// Mitsubishi GX Works2 project: halvanika_new3   PLC: FX3U/FX3UC

TYPE vat : STRUCT
  entire : INT;
  prioriyry : BOOL;
  timer_s : DINT;
  on_off : BOOL;
  timer_off : BOOL;
  timer_real : DINT;
  vibor : INT;
  air_off : BOOL;
  vanna_off : BOOL;
END_STRUCT END_TYPE

// global labels: Global1
VAR_GLOBAL
  incFR AT D100 : INT;  (* позиция балки по ваннам *)
  incUD AT D101 : INT;  (* позиция балки по вертикали *)
  muving AT D102 : INT;  (* управление с HMI балкой *)
  Program_exec AT D103 : INT;  (* переключение режимов работы *)
  tub : ARRAY [0..15] OF vat;  (* массив структуры ванн *)
  init_reset AT M100 : BOOL;  (* переключение инициализации *)
  autoStop AT D104 : INT;  (* включение окна ошибок *)
  text AT D105 : STRING[32];  (* Сообщения об ошибках *)
  TEST_ONOFF AT D107 : INT;  (* Тестовое отключение бурбуляторов *)
  Hide_button AT D108 : INT;
  temper AT D110 : ARRAY [0..8] OF INT;
  load_z AT D120 : INT;
  upload_z AT D121 : INT;
  init_move : BOOL;
  reset_timers : BOOL;
  pause AT D122 : INT;
  blink_botton AT D123 : INT;
  ch AT D124 : INT;
END_VAR

// task Task_01 (event TRUE, interval 0, priority 31): Init

PROGRAM Init
VAR
  Manual_1 : Manual;
  Auto_1 : Auto;
  Reset_1 : Reset;
  init : BOOL;
  Stop_program : BOOL;
  Count : INT;
  blink : TON;
  TR1 : R_TRIG;
  Count2 : INT;
  bath_02 : TON;
  bath_03 : TON;
  bath_04 : TON;
  bath_05 : TON;
  bath_06 : TON;
  bath_07 : TON;
  bath_08 : TON;
  bath_09 : TON;
  bath_10 : TON;
  bath_11 : TON;
  bath_12 : TON;
  bath_13 : TON;
  bath_14 : TON;
END_VAR
(*------------------------------INIT----------------------------------------------------*)
IF NOT init THEN
	incFR := 1;
	incUD := -1;
	Hide_button := 1;
	Program_exec := 0;
	muving := 0;
	TEST_ONOFF :=1;
reset_timers := FALSE;
pause := 0;
blink_botton := 0;

	tub[1].prioriyry := 0;
	tub[2].prioriyry := 1;
	tub[3].prioriyry := 0;
	tub[4].prioriyry := 0;
	tub[5].prioriyry := 1;
	tub[6].prioriyry := 0;
	tub[7].prioriyry := 0;
	tub[8].prioriyry := 1;
	tub[9].prioriyry := 0;
	tub[10].prioriyry := 1;
	tub[11].prioriyry := 1;
	tub[12].prioriyry := 0;
	tub[13].prioriyry := 0;
	tub[14].prioriyry := 1;
	tub[15].prioriyry := 1;
	
		FOR Count := 1 TO 15 DO
			tub[Count].vanna_off := 1;
			tub[Count].air_off := 0;
		END_FOR;	
	
	init := TRUE;
END_IF;

(*------------------------------PROGAM----------------------------------------------------*)

IF (X000 = 0) AND (X001 = 1) AND (X002 = 1) THEN incFR := 1;  END_IF;
IF (X000 = 1) AND (X001 = 1) AND (X002 = 1) THEN incFR := 15; END_IF;
IF (X004 = 1)  THEN incUD := -1; ELSIF  (X003 = 1) THEN  incUD := 1;  END_IF;
IF incFR < 1 OR incFR > 15 THEN autoStop := 1; END_IF;
	
(*------------------------------Timers----------------------------------------------------*)

	FOR count:=2 TO 14 DO
		IF NOT tub[Count].timer_off THEN tub[Count].timer_real:=0; END_IF;
	END_FOR;
	
IF Program_exec <> 3 THEN	
bath_02(IN:= INT_TO_BOOL(tub[2].entire) ,PT:= DINT_TO_TIME(tub[2].timer_s) * 1000);
bath_03(IN:= INT_TO_BOOL(tub[3].entire) ,PT:= DINT_TO_TIME(tub[3].timer_s) * 1000);
bath_04(IN:= INT_TO_BOOL(tub[4].entire) ,PT:= DINT_TO_TIME(tub[4].timer_s) * 1000);
bath_05(IN:= INT_TO_BOOL(tub[5].entire) ,PT:= DINT_TO_TIME(tub[5].timer_s) * 1000);
bath_06(IN:= INT_TO_BOOL(tub[6].entire) ,PT:= DINT_TO_TIME(tub[6].timer_s) * 1000);
bath_07(IN:= INT_TO_BOOL(tub[7].entire) ,PT:= DINT_TO_TIME(tub[7].timer_s) * 1000);
bath_08(IN:= INT_TO_BOOL(tub[8].entire) ,PT:= DINT_TO_TIME(tub[8].timer_s) * 1000);
bath_09(IN:= INT_TO_BOOL(tub[9].entire) ,PT:= DINT_TO_TIME(tub[9].timer_s) * 1000);
bath_10(IN:= INT_TO_BOOL(tub[10].entire) ,PT:= DINT_TO_TIME(tub[10].timer_s) * 1000);
bath_11(IN:= INT_TO_BOOL(tub[11].entire) ,PT:= DINT_TO_TIME(tub[11].timer_s) * 1000);
bath_12(IN:= INT_TO_BOOL(tub[12].entire) ,PT:= DINT_TO_TIME(tub[12].timer_s) * 1000);
bath_13(IN:= INT_TO_BOOL(tub[13].entire) ,PT:= DINT_TO_TIME(tub[13].timer_s) * 1000);
bath_14(IN:= INT_TO_BOOL(tub[14].entire) ,PT:= DINT_TO_TIME(tub[14].timer_s) * 1000);

tub[2].timer_off := NOT bath_02.Q; tub[2].timer_real := TIME_TO_DINT(bath_02.ET) / 1000;
tub[3].timer_off := NOT bath_03.Q; tub[3].timer_real := TIME_TO_DINT(bath_03.ET) / 1000;
tub[4].timer_off := NOT bath_04.Q; tub[4].timer_real := TIME_TO_DINT(bath_04.ET) / 1000;
tub[5].timer_off := NOT bath_05.Q; tub[5].timer_real := TIME_TO_DINT(bath_05.ET) / 1000;
tub[6].timer_off := NOT bath_06.Q; tub[6].timer_real := TIME_TO_DINT(bath_06.ET) / 1000;
tub[7].timer_off := NOT bath_07.Q; tub[7].timer_real := TIME_TO_DINT(bath_07.ET) / 1000;
tub[8].timer_off := NOT bath_08.Q; tub[8].timer_real := TIME_TO_DINT(bath_08.ET) / 1000;
tub[9].timer_off := NOT bath_09.Q; tub[9].timer_real := TIME_TO_DINT(bath_09.ET) / 1000;
tub[10].timer_off := NOT bath_10.Q; tub[10].timer_real := TIME_TO_DINT(bath_10.ET) / 1000;
tub[11].timer_off := NOT bath_11.Q; tub[11].timer_real := TIME_TO_DINT(bath_11.ET) / 1000;
tub[12].timer_off := NOT bath_12.Q; tub[12].timer_real := TIME_TO_DINT(bath_12.ET) / 1000;
tub[13].timer_off := NOT bath_13.Q; tub[13].timer_real := TIME_TO_DINT(bath_13.ET) / 1000;
tub[14].timer_off := NOT bath_14.Q; tub[14].timer_real := TIME_TO_DINT(bath_14.ET) / 1000;

(* Включить ток*);
IF tub[5].entire = 1 THEN Y013 := INT_TO_BOOL(TEST_ONOFF); END_IF;
IF tub[10].entire = 1 THEN Y024 :=  INT_TO_BOOL(TEST_ONOFF); END_IF;
IF tub[11].entire = 1 THEN Y014 :=  INT_TO_BOOL(TEST_ONOFF); END_IF;
(* Выключить ток*);
IF NOT tub[5].timer_off THEN Y013 := 0; END_IF;
IF NOT tub[10].timer_off THEN Y024 := 0; END_IF;
IF NOT tub[11].timer_off THEN Y014 := 0; END_IF;
	
(* Включить спрей*)
IF tub[3].on_off THEN Y016 := INT_TO_BOOL(TEST_ONOFF); ELSE Y016 := FALSE; END_IF;
IF tub[6].on_off THEN Y017 :=  INT_TO_BOOL(TEST_ONOFF); ELSE Y017 := FALSE; END_IF;
IF tub[9].on_off THEN Y020 :=  INT_TO_BOOL(TEST_ONOFF); ELSE Y020 := FALSE; END_IF;
IF tub[12].on_off THEN Y021 :=  INT_TO_BOOL(TEST_ONOFF); ELSE Y021 := FALSE; END_IF;

(* Включить спрей
IF tub[3].entire = 1 THEN Y016 :=  INT_TO_BOOL(TEST_ONOFF); END_IF;
IF tub[6].entire = 1 THEN Y017 :=  INT_TO_BOOL(TEST_ONOFF); END_IF;
IF tub[9].entire = 1 THEN Y020 :=  INT_TO_BOOL(TEST_ONOFF); END_IF;
IF tub[12].entire = 1 THEN Y021 :=  INT_TO_BOOL(TEST_ONOFF); END_IF;

Выключить спрей
IF NOT tub[3].timer_off THEN Y016 := 0; END_IF;
IF NOT tub[6].timer_off THEN Y017 := 0; END_IF;
IF NOT tub[9].timer_off THEN Y020 := 0; END_IF;
IF NOT tub[12].timer_off THEN Y021 := 0; END_IF;
	
Выключить сушку
IF NOT tub[14].timer_off THEN Y011 := 0;  END_IF; 
*);
END_IF;

IF reset_timers THEN
	bath_02(IN:= FALSE);
	bath_03(IN:= FALSE);
	bath_04(IN:= FALSE);
	bath_05(IN:= FALSE);
	bath_06(IN:= FALSE);
	bath_07(IN:= FALSE);
	bath_08(IN:= FALSE);
	bath_09(IN:= FALSE);
	bath_10(IN:= FALSE);
	bath_11(IN:= FALSE);
	bath_12(IN:= FALSE);
	bath_13(IN:= FALSE);
	bath_14(IN:= FALSE);
	reset_timers := FALSE;
END_IF;

(*------------------------------CASE----------------------------------------------------*)

IF pause = 0 AND (Program_exec = 1 OR  (X011 = 1)) THEN
	Manual_1(); 
	
ELSIF Program_exec = 2 THEN
	Auto_1(); 
	(* -------------Air Pump----------*)
	Y030 := tub[2].air_off;
	Y031 := tub[3].air_off;
	Y032 := tub[4].air_off;
	Y033 := tub[5].air_off;
	Y034 := tub[6].air_off;
	Y035 := tub[7].air_off;
	Y036 := tub[8].air_off;
	Y037 := tub[9].air_off;
	Y040 := tub[10].air_off;
	Y041 := tub[11].air_off;
	Y042 := tub[12].air_off;
	Y043 := tub[13].air_off;
	
ELSIF Program_exec = 3 THEN
	Reset_1();
	reset_timers := TRUE;
END_IF;

IF pause = 1 AND (Program_exec = 1 OR  (X011 = 1)) THEN
	Program_exec := 2;
	pause := 2;
	END_IF;
muving := 0;


(*------------------------------STOP----------------------------------------------------*)

IF (X013 = 1) OR (X021 = 1) OR (X012 = 1)  OR autoStop = 1THEN
	Program_exec := 0;
	muving := 0;
	autoStop := 0;
	Hide_button := 0;
	pause := 0;

	Y000 :=0;	Y010 :=0;	Y020 :=0;
	Y001 :=0;	Y011 :=0;	Y021 :=0;
	Y002 :=0;	Y012 :=0;	Y022 :=0;
	Y003 :=0;	Y013 :=0;	Y023 :=0;
	Y004 :=0;	Y014 :=0;	Y024 :=0;
	Y005 :=0;	Y015 :=0;	Y025 :=0;
	Y006 :=0;	Y016 :=0;	Y026 :=0;
	Y007 :=0;	Y017 :=0;	Y027 :=0;
		(* -------------Air Pump----------*)
	Y030 := 0;	Y040 := 0;
	Y031 := 0;	Y041 := 0;
	Y032 := 0;	Y042 := 0;
	Y033 := 0;	Y043 := 0;
	Y034 := 0;	Y044 := 0;
	Y035 := 0;	Y045 := 0;
	Y036 := 0;	Y046 := 0;
	Y037 := 0;	Y047 := 0;
	
	reset_timers := TRUE;
	
		FOR Count := 1 TO 15 DO
			tub[Count].timer_off  := 0;
			tub[Count].timer_real := 0;
			tub[Count].on_off := 0;
			tub[Count].air_off := 0;
		END_FOR;	
		
		init_move:= FALSE; 
		init_reset := FALSE;
		

END_IF;
END_PROGRAM

FUNCTION_BLOCK Auto
VAR
  blink : TON;
  init : BOOL;
  vanna : INT;
  Count : INT;
  vanna1 : INT;
  tabs : INT;
  TR1 : R_TRIG;
  Err : INT;
  prime : BOOL;
  vanna15 : INT;
  moving_1 : moving;
  pause_t : TON;
  TR2 : R_TRIG;
  stopd : BOOL;
  vanOff : INT;
  Counts : INT;
END_VAR
(*------------------------------INIT----------------------------------------------------*)
IF NOT init_reset THEN
	text:= "";
	IF incUD = 1 THEN text:= "Lower the beam down"; Program_exec := 0; END_IF; 
		vanna1 := 0;
		vanna := 0;
		vanna15 := 0;
		pause := 1;
		stopd := FALSE;
		ch := 1;
		vanOff := 1;
		(*Doors close*)
		Y022 := 0;
		blink_botton := 2;
		pause_t(IN := FALSE);
		TR2(_CLK := FALSE);
	init_reset :=TRUE;
	
END_IF;


(*------------------------------Blink----------------------------------------------------*)
Y026:= 0;
blink(IN:= NOT blink.Q, PT:= T#1s);
TR1(_CLK:= blink.Q );
IF TR1.Q THEN
	Y015:= NOT Y015;
	IF  tub[15].entire = 1 AND upload_z = 0 THEN Y027:= NOT Y027; ELSE Y027:= FALSE; END_IF;
END_IF;

(*------------------------------Blink----------------------------------------------------*)

pause_t (IN:= stopd, PT:= T#4s);
TR2(_CLK:= pause_t.Q );
IF TR2.Q THEN
	tabs:= tabs +1;
	stopd := FALSE;
END_IF;

(*-----------------------------CICLE-----------------------------------------------------*)


IF X006 = 1 OR upload_z = 1 THEN vanna15 := 15; upload_z := 1; END_IF;
IF  X005 = 1 OR load_z = 1 THEN vanna1 := 1; tub[1].entire := 1; load_z := 1; END_IF;
	
IF vanna = 0 THEN
	prime := FALSE;
	tabs := 0;
	vanOff := 1;
	Counts := 0;
	
	FOR Count := 2 TO 14 BY 1 DO
		IF tub[Count].entire = 1 AND tub[Count+vanOff ].entire = 0 AND NOT tub[Count].timer_off AND NOT tub[Count].prioriyry AND NOT prime THEN vanna := Count; prime := FALSE;  END_IF;
		IF tub[Count].entire = 1 AND tub[Count+vanOff ].entire = 0 AND NOT tub[Count].timer_off AND tub[Count].prioriyry THEN vanna := Count; prime := TRUE; END_IF;
	END_FOR;	
	
	IF tub[1].entire =0 AND  vanna15 = 15 THEN vanna := vanna15; END_IF;
	IF tub[2].entire =0 AND vanna1 = 1 THEN vanna := vanna1; END_IF;
	
	FOR Count := vanna TO 14 DO
		IF tub[vanna+vanOff ].vanna_off = 0 THEN vanOff := vanOff + 1;
		ELSE
			EXIT;
		END_IF;
	END_FOR;
	 IF tub[vanna+vanOff].entire = 1 THEN vanna := 0; END_IF;
	
END_IF;
		
(*-----------------------------ERROR-----------------------------------------------------*)	
(*	Ошибки обрабатываем в HMI *)
(*-----------------------------ERROR-----------------------------------------------------*)		
	
	IF vanna > 0 AND tabs = 0 THEN			
				IF incFR > vanna THEN
					moving_1(mv:=  2 ,mv_change:= incFR - vanna ,incount:= incFR, incUP:= incUD, ends:= tabs);
				ELSIF  incFR < vanna THEN
					moving_1(mv:=  1 ,mv_change:= vanna - incFR ,incount:= incFR, incUP:= incUD, ends:= tabs);
				ELSE
					tabs:= 1;
				END_IF;
		
	ELSE
 
	    CASE vanna OF
	
			1:  IF tub[vanna+vanOff].entire = 0 THEN
			CASE tabs OF	
						1: moving_1(mv:=  3 ,mv_change:= 1 ,incount:= incFR, incUP:= incUD, ends:= tabs);
						2: IF TRUE THEN tub[vanna].entire := 0; tabs:= tabs+1; END_IF;
						3: tabs:= tabs +1;
						4: moving_1(mv:= 1 ,mv_change:= vanOff ,incount:= incFR, incUP:= incUD, ends:= tabs);
						5: IF TRUE THEN stopd := TRUE; tub[vanna+vanOff].air_off := TRUE; END_IF;
						6: moving_1(mv:=  4 ,mv_change:= 1 ,incount:= incFR, incUP:= incUD, ends:= tabs);
						7: tabs:= tabs +1;
						8: IF TRUE THEN
							tub[vanna+vanOff].entire := 1;
							tub[vanna+vanOff].timer_off := TRUE;
							vanna := 0;
							vanna1 := 0;
							tabs:= 0;
							END_IF;
			END_CASE;
			END_IF;
		
			3, 6, 9, 12:  IF TRUE THEN
			CASE tabs OF
						1: IF TRUE THEN tub[vanna].on_off := TRUE; tabs:= tabs+1; END_IF;	
						2: moving_1(mv:=  3 ,mv_change:= 1 ,incount:= incFR, incUP:= incUD, ends:= tabs);
						3: IF TRUE THEN tub[vanna].entire := 0; tub[vanna].air_off := FALSE; tub[vanna].on_off := FALSE; tabs:= tabs+1; END_IF;
						4: moving_1(mv:= 1 ,mv_change:= vanOff ,incount:= incFR, incUP:= incUD, ends:= tabs); 
						5: IF TRUE THEN stopd := TRUE; tub[vanna+vanOff].air_off := TRUE; END_IF;
						6: moving_1(mv:=  4 ,mv_change:= 1 ,incount:= incFR, incUP:= incUD, ends:= tabs);
						7: tabs:= tabs +1;
						8: IF TRUE THEN
								tub[vanna+vanOff].entire := 1;
								tub[vanna+vanOff].timer_off := TRUE;
								vanna := 0;
								tabs:= 0;
							END_IF;
			END_CASE;
			END_IF;
	
			2, 4, 5, 8, 10, 11:  IF TRUE THEN
			CASE tabs OF	
						1: moving_1(mv:=  3 ,mv_change:= 1 ,incount:= incFR, incUP:= incUD, ends:= tabs);
						2: IF TRUE THEN tub[vanna].entire := 0; tub[vanna].air_off := FALSE; tabs:= tabs+1; END_IF;
						3: tabs:= tabs +1;
						4: moving_1(mv:= 1 ,mv_change:= vanOff ,incount:= incFR, incUP:= incUD, ends:= tabs); 
						5: IF TRUE THEN stopd := TRUE; tub[vanna+vanOff].air_off := TRUE; END_IF;
						6: moving_1(mv:=  4 ,mv_change:= 1 ,incount:= incFR, incUP:= incUD, ends:= tabs);
						7: tabs:= tabs +1;
						8: IF TRUE THEN
							tub[vanna+vanOff].entire := 1;
							tub[vanna+vanOff].timer_off := TRUE;
								vanna := 0;
								tabs:= 0;
							END_IF;
			END_CASE;
			END_IF;
	
			7:  IF tub[vanna+vanOff +1].entire = 0 THEN
			CASE tabs OF	
						1: moving_1(mv:=  3 ,mv_change:= 1 ,incount:= incFR, incUP:= incUD, ends:= tabs);
						2: IF TRUE THEN tub[vanna].entire := 0; tub[vanna].air_off := FALSE; tabs:= tabs+1; END_IF;
						3: tabs:= tabs +1;
						4: moving_1(mv:= 1 ,mv_change:= vanOff ,incount:= incFR, incUP:= incUD, ends:= tabs); 
						5: IF TRUE THEN stopd := TRUE; tub[vanna+vanOff].air_off := TRUE; END_IF;
						6: moving_1(mv:=  4 ,mv_change:= 1 ,incount:= incFR, incUP:= incUD, ends:= tabs);
						7: tabs:= tabs +1;
						8: IF TRUE THEN
							tub[vanna+vanOff].entire := 1;
							tub[vanna+vanOff].timer_off := TRUE;
							tabs:=tabs+1;
							END_IF;
						9:	IF NOT tub[vanna+vanOff].timer_off  THEN
								vanna := vanna + 1;
								tabs:= 0;
							END_IF;
							
			END_CASE;
			END_IF;
	
			13:  IF TRUE THEN
			CASE tabs OF	
						1: moving_1(mv:=  3 ,mv_change:= 1 ,incount:= incFR, incUP:= incUD, ends:= tabs);
						2: IF TRUE THEN tub[vanna].entire := 0; tub[vanna].air_off := FALSE; tabs:= tabs+1; END_IF;
						3: tabs:= tabs +1;
						4: moving_1(mv:= 1 ,mv_change:= vanOff ,incount:= incFR, incUP:= incUD, ends:= tabs); 
						(*Doors open*)
						5: IF TRUE THEN Y022 := 1; tabs:= tabs+1; END_IF;
						6: moving_1(mv:=  4 ,mv_change:= 1 ,incount:= incFR, incUP:= incUD, ends:= tabs);
						7: tabs:= tabs +1;
						8: IF TRUE THEN
						(*Doors close*)
							Y022 := 0;
							tub[vanna+vanOff].entire := 1;
							tub[vanna+vanOff].timer_off := TRUE;
							vanna := 0;
							tabs:= 0;
							END_IF;
			END_CASE;
			END_IF;
			
			14:  IF TRUE THEN
			CASE tabs OF
						(*-Doors open-вернуться*)	
						1: IF TRUE THEN Y022 := 1; tabs:= tabs+1; END_IF;
						2: moving_1(mv:=  3 ,mv_change:= 1 ,incount:= incFR, incUP:= incUD, ends:= tabs);
						3: tabs:= tabs +1;
						4: IF TRUE THEN Y022:=0; tub[vanna].entire := 0; tabs:= tabs+1; END_IF;
						5: moving_1(mv:= 1 ,mv_change:= 1 ,incount:= incFR, incUP:= incUD, ends:= tabs);
						6: moving_1(mv:=  4 ,mv_change:= 1 ,incount:= incFR, incUP:= incUD, ends:= tabs);
						7: tabs:= tabs +1;
						8: IF TRUE THEN
							tub[vanna+1].entire := 1;
							tub[vanna+1].timer_off := TRUE;
							vanna := 0;
							tabs:= 0;
							END_IF;
			END_CASE;
			END_IF;
			
			15:  IF tub[1].entire = 0 THEN
			CASE tabs OF	
						1: moving_1(mv:=  3 ,mv_change:= 1 ,incount:= incFR, incUP:= incUD, ends:= tabs);
						2: IF TRUE THEN tub[vanna].entire := 0; tabs:= tabs+1; END_IF;
						3: moving_1(mv:= 2 ,mv_change:= 14 ,incount:= incFR, incUP:= incUD, ends:= tabs);
						4: moving_1(mv:=  4 ,mv_change:= 1 ,incount:= incFR, incUP:= incUD, ends:= tabs);
						5: tabs:= tabs +2;
						7: IF TRUE THEN
							vanna := 0;
							vanna15 :=0;
							tabs:= 0;
							END_IF;
			END_CASE;
			END_IF;
		
	    END_CASE;
    END_IF;

IF vanna = 0 AND pause = 2 THEN  pause := 0; Program_exec := 1; ELSE  Program_exec := 2;  END_IF;
END_FUNCTION_BLOCK

FUNCTION_BLOCK Manual
VAR
  blink : TON;
  TR1 : R_TRIG;
  tabs : INT;
  MV : INT;
  DELTA_MV : INT;
  moving_1 : moving;
END_VAR

Y015 := 0;
blink(IN:= NOT blink.Q, PT:= T#1s);
TR1(_CLK:= blink.Q );
IF TR1.Q THEN
	Y026:= NOT Y026;
END_IF;
pause := 0;
blink_botton := 1;
Program_exec := 1;
IF  (X001 = 0)  THEN ch:=0; ELSE ch:=1; END_IF;
DELTA_MV:= 1;
init_reset := FALSE;

	IF		((X005 = 1) OR (muving=1))  AND  (incFR < 15) THEN
		MV:= 1;					(* Forward *)
	ELSIF ((X006 = 1) OR (muving=2)) AND  (incFR > 1) THEN
		MV:= 2;						(* Revers *)
	ELSIF ((X007 = 1) OR (muving=3)) THEN
		MV:= 3;					(* Up *)
	ELSIF ((X010 = 1)  OR (muving=4)) THEN
		MV:= 4;						(* Down *)
	END_IF;
	moving_1(mv:=  MV, mv_change:= DELTA_MV, incount:= incFR, incUP:= incUD);
muving := 0;
MV:=0;
END_FUNCTION_BLOCK

FUNCTION_BLOCK Reset
VAR
  Count : INT;
  init : BOOL;
END_VAR
IF (X000 = 0) AND (X001 = 1) AND (X002 = 1) THEN incFR := 1; END_IF;
IF (X000 = 1) AND (X001 = 1) AND (X002 = 0) THEN incFR := 15; END_IF;
IF (X004 = 1)  THEN incUD := -1; ELSIF  (X003 = 1) THEN  incUD := 1;  END_IF;
	
(*------------------------------INIT----------------------------------------------------*)
	IF NOT init THEN 
	Y027 :=1;	
	Y000 :=0;	Y010 :=0;	Y020 :=0;
	Y001 :=0;	Y011 :=0;	Y021 :=0;
	Y002 :=0;	Y012 :=0;	Y022 :=0;
	Y003 :=0;	Y013 :=0;	Y023 :=0;
	Y004 :=0;	Y014 :=0;	Y024 :=0;
	Y005 :=0;	Y015 :=0;	Y025 :=0;
	Y006 :=0;	Y016 :=0;	Y026 :=0;
	Y007 :=0;	Y017 :=0;	
		(* -------------Air Pump----------*)
	Y030 := 0;	Y040 := 0;
	Y031 := 0;	Y041 := 0;
	Y032 := 0;	Y042 := 0;
	Y033 := 0;	Y043 := 0;
	Y034 := 0;	Y044 := 0;
	Y035 := 0;	Y045 := 0;
	Y036 := 0;	Y046 := 0;
	Y037 := 0;	Y047 := 0;
	
	tub[1].prioriyry := 0;
	tub[2].prioriyry := 1;
	tub[3].prioriyry := 0;
	tub[4].prioriyry := 0;
	tub[5].prioriyry := 1;
	tub[6].prioriyry := 0;
	tub[7].prioriyry := 0;
	tub[8].prioriyry := 1;
	tub[9].prioriyry := 0;
	tub[10].prioriyry := 1;
	tub[11].prioriyry := 1;
	tub[12].prioriyry := 0;
	tub[13].prioriyry := 0;
	tub[14].prioriyry := 1;
	tub[15].prioriyry := 1;
	
	muving := 0;
blink_botton := 3;
	init := TRUE; 
	END_IF;
	
	init_reset := FALSE;
	pause := 0;
	
	FOR Count := 1 TO 15 DO
		tub[Count].entire := 0;
		tub[Count].timer_off  := 0;
		tub[Count].timer_real:=0;
		tub[Count].on_off:=0;
		tub[Count].vanna_off := 1;
		tub[Count].air_off := 0;
	END_FOR;	
 
 (*IF X004 = 0 THEN moving_1(mv:=  4, mv_change:= 1, incount:= incFR, incUP:= incUD); END_IF;*)
 	
 	IF (X000 = 0) AND (X001 = 1) AND (X002 = 1) THEN
		Y000 := 0;
		Y001 := 0;
		Y002 := 0;
		Y003 := 0;
		Y004 := 0;
		incFR := 1; 
	Program_exec := 0;
		Y027 :=0;
 	ELSE
 		Y004 := 1;
		Y002 := 0;
		Y001 := 1;
		IF (X002 = 1) THEN Y003 := 0; 
		ELSIF (X001 = 1) AND (X002 = 0) THEN Y003 := 1; 
		END_IF;
		
END_IF;
END_FUNCTION_BLOCK

FUNCTION_BLOCK moving
VAR_INPUT
  mv : INT;
END_VAR
VAR
  flag : INT;
  temp : INT;
END_VAR
VAR_INPUT
  mv_change : INT;
END_VAR
VAR
  change : INT;
  beg : INT;
END_VAR
VAR_IN_OUT
  incount : INT;
END_VAR
VAR
  count : INT;
END_VAR
VAR_IN_OUT
  incUP : INT;
END_VAR
VAR_OUTPUT
  ends : INT;
END_VAR
VAR
  init : BOOL;
END_VAR
	(*------------------------------INIT----------------------------------------------------*)
IF NOT init_move THEN
	flag :=0;
	temp:=0;
	
				incount := incount;
			incUP:=incUP;
			beg:=1;

	init_move:=TRUE;
	END_IF;
	
	IF temp = 0  AND mv <> 0 AND mv_change <> 0 THEN
		flag := 1; 
		temp := mv;
		change := mv_change-ch; 
		ch:=1;
		beg := 1;

	END_IF;

	CASE temp OF
			1:		IF flag = 1 THEN 
						Y000 := 1;
						Y003 := 0;
						Y004 := 1;
					IF (X000 = 1) AND flag =1THEN change := change - beg; 
							incount := incount +beg;
							beg := 0;
							Y002 := 1;
						ELSE 
							beg :=1;
							 END_IF;
						IF change <= 0 THEN 	flag := 2; END_IF;
					ELSIF (X000 = 0) AND (X001 = 0) AND (X002 = 1) AND flag = 2  THEN
						Y003 := 1;
						Y002 := 0;	
				(*			REPEAT
								IF (X001 = 1) THEN change := change - 1; moveFR := 1;END_IF;
							UNTIL change = 0 END_REPEAT; *)
						flag := 3;
					ELSIF (X000 = 1) AND (X001 = 0) AND (X002 = 0)  AND flag = 3 THEN
						Y002 := 0;
						Y003 := 0;
						flag := 4;
					ELSIF (X001 = 1) AND (X002 = 0)  AND flag = 4  THEN
						Y000 := 0;
						Y002 := 0;
						Y003 := 0;
						flag := 0;
						temp := 0;
						Y004 := 0;
incount := incount+1;
ends:= 1+ends;
						END_IF;

			(*-----------------*)
			2:		IF flag = 1 THEN 
						Y001 := 1;
						Y003 := 0;
						Y004 := 1;
					IF (X002 = 1) AND flag =1THEN change := change - beg; 
							incount := incount -beg;
							beg := 0;
							Y002 := 1;
						ELSE 
							beg :=1;
							 END_IF;
						IF change <= 0 THEN 	flag := 2; END_IF;
					ELSIF  (X000 = 1) AND (X001 = 0) AND (X002 = 0)  AND flag = 2 THEN
						Y003 := 1;
						Y002 := 0;
						flag := 3;
					ELSIF (X000 = 0) AND (X001 = 0) AND (X002 = 1)   AND flag = 3 THEN
						Y002 := 0;
						Y003 := 0;
						flag := 4;
					ELSIF  (X000 = 0) AND (X001 = 1)  AND flag = 4  THEN
						Y001 := 0;
						Y002 := 0;
						Y003 := 0;
						flag := 0;
						temp := 0;
						Y004 := 0;
ends:= 1+ends;				
incount := incount-1;	
						END_IF;
						
						3:		IF  (X003 = 1) THEN 
						Y000 := 0;
						Y001 := 0;
						Y002 := 0;
						Y003 := 0;
						Y005 := 0;
						temp := 0; 
						incUP:= 1;
ends:= 1+ends;
					ELSE
						Y000 := 1;
						Y002 := 0;
						IF Program_exec = 2 AND (incount = 3 OR incount = 6 OR incount = 9 OR incount = 12) THEN Y003 := 0; ELSE Y003 := 1; END_IF;
						Y005 := 1;
					END_IF;
			(*-----------------*)		
			4:		IF (X004 = 1)  THEN 
						Y000 := 0;
						Y001 := 0;
						Y002 := 0;
						Y003 := 0;
						Y005 := 0;
						temp := 0; 
						incUP:= -1;
ends:= 1+ends;
					ELSE
						Y001 := 1;
						Y002 := 0;
						IF Program_exec = 2 AND (incount  > 1 AND incount < 14) THEN Y003 := 0; ELSE Y003 := 1; END_IF;
						Y005 := 1;
					END_IF;
		
			ELSE
			incount := incount;
			incUP:=incUP;
			flag := 0;
			ends:=0;
					temp := 0;
	END_CASE;
END_FUNCTION_BLOCK
